FUNCTION_BLOCK FB_Stop
VAR_INPUT
(*È«¾Ö*)
	Mode:DINT;
	PowerState:BOOL;
	(*BCGapMode*)
	BCGapStop:BOOL;
END_VAR
VAR_OUTPUT
	FbID:DINT:=1001;

	BCGapState:DINT;
	BCGapBusy:BOOL;
	BCGapDone:BOOL;

	Error:BOOL;
	ErrorID:DINT;
END_VAR
VAR
	PhaseShifterLin_MC_Stop: MC_Stop;
	fb_ton: TON;
	fb_ton1: TON;
	fb_ton2: TON;
	fb_ton_debug_1:TON;
	fb_ton_debug_2:TON;
	fb_ton_debug_3:TON;
	fb_ton_debug_4:TON;
	fb_ton_BC: TON;

END_VAR

IF PowerState=1 THEN
	IF Mode=1 AND BCGapStop THEN
		A_BCGapStop();
	ELSE
		FB_PlcEmergencyStop();
	END_IF
END_IF

ACTION A_BCGapStop:
IF BCGapStop THEN
BCGapBusy:=TRUE;
BCGapDone:=FALSE;
fb_ton_BC(PT:=t#100ms);
A_StopMC();
CASE BCGapState OF
	0:
		IF PhaseShifterLin_MC_Stop.Error  THEN
			ErrorID:=1;
			BCGapState:=-100;
			PhaseShifterLin_MC_Stop.Execute:=FALSE;
			A_StopMC();
		ELSE
			BCGapState:=1;
		END_IF
	1:
		PhaseShifterLin_MC_Stop.Execute:=TRUE;
		fb_ton_BC.IN:=TRUE;
		BCGapState:=2;
	2:
		IF  NOT PhaseShifterLin_MC_Stop.Done  THEN
				BCGapState:=2;
		ELSE
			BCGapState:=88;
			PhaseShifterLin_MC_Stop.Execute:=FALSE;
			A_StopMC();
		END_IF

	88:
		BCGapStop:=FALSE;
		BCGapState:=0;
		BCGapBusy:=FALSE;
		BCGapDone:=TRUE;
		Error:=FALSE;
		ErrorID:=0;
		fb_ton_BC.IN:=FALSE;

	-100:
		FB_PlcEmergencyStop();
		BCGapStop:=FALSE;
		BCGapState:=-100;
		BCGapBusy:=FALSE;
		BCGapDone:=FALSE;
		Error:=TRUE;
		PhaseShifterLin_MC_Stop.Execute:=FALSE;
		A_StopMC();
		fb_ton_BC.IN:=FALSE;

END_CASE
END_IF
END_ACTION

ACTION A_StopMC:
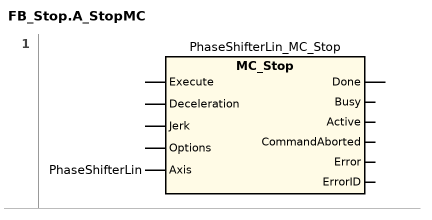
// NETWORK 1
PhaseShifterLin_MC_Stop(Axis := PhaseShifterLin); // MC_Stop
END_ACTION

END_FUNCTION_BLOCK

(* stored: Version 1.1.0.1, ProductVersion 3.1.4024.6
   POU FB_Stop: Id {3e354bcb-4e4f-4b34-9851-51b9542d0760}, SpecialFunc None
   Action A_BCGapStop: Id {09d39807-0cc9-4816-a94c-73c13504c1f7}
   Action A_StopMC: Id {b171a3f0-94b4-4ac2-92c0-8ca964cc4005} *)
